FUNCTION TryConvert_UINT_TO_BOOL : BOOL
VAR_INPUT
	in : UINT;
	out : REFERENCE TO BOOL;
END_VAR

out := UINT_TO_BOOL(in);
TryConvert_UINT_TO_BOOL := TRUE;

END_FUNCTION

(* stored: Version 1.1.0.1, ProductVersion 3.1.4024.12
   POU TryConvert_UINT_TO_BOOL: Id {02e75eca-cc87-49f7-a04a-e6057abe5ed8}, SpecialFunc None *)
